{attribute 'TcGenerated'}
{attribute 'no-analysis'}
{attribute 'linkalways'}
// This function has been automatically generated from the project information.
VAR_GLOBAL CONSTANT
	{attribute 'const_non_replaced'}
	stLibVersion_EfficientIO_Communicator : ST_LibVersion := (iMajor := 2, iMinor := 1, iBuild := 0, iRevision := 0, nFlags := 0, sVersion := '2.1');
END_VAR

(* stored: Version 1.1.0.1, ProductVersion 3.1.4024.11
   GVL Global_Version: Id {21963910-1e7f-48b6-a92d-24ac6377e96a} *)
